{attribute 'qualified_only'}
{attribute 'strict'}
TYPE E_EasyTempState :
(
	Stopped := 0,
	Running := 1,
	Tuning := 2,
	Resetting := 99
);
END_TYPE

(* stored: Version 1.1.0.1, ProductVersion 3.1.4024.12
   DUT E_EasyTempState: Id {96a487c9-00ef-4f02-94af-7625d13c80b4} *)
